{attribute 'strict'}
TYPE E_VisuCtrlPageState :
(
	SCREEN_UNINITIALIZED 		:= 0,	(*  *)
	SCREEN_INITIALIZING 		:= 1,	(*  *)
	SCREEN_READY_INITIALIZED	:= 2,	(*  *)
	SCREEN_AUTO					:= 3,	(*  *)
	SCREEN_MODE_CHANGE			:= 4,	(*  *)
	SCREEN_MANUAL_CYLINDERS		:= 5,	(*  *)
	SCREEN_MANUAL_MOTORS		:= 6,	(*  *)
	//SCREEN_MANUAL_SAFETY		:= 7,	(*  *)
	SCREEN_MANUAL_INPUTS		:= 7,	(*  *)
	SCREEN_MANUAL_OUTPUTS		:= 8,	(*  *)
	SCREEN_MANUAL_ROBOTS		:= 9,	(*  *)
	SCREEN_MANUAL_OTHERS		:= 10,	(*  *)
	SCREEN_ALARMS				:= 11,	(*  *)
	SCREEN_RECIPES				:= 12,	(*  *)
	SCREEN_RESET				:= 13,	(*  *)
	SCREEN_ABORTING				:= 14,	(*  *)
	SCREEN_EMERGENCY			:= 15	(*  *)
);
END_TYPE

(* stored: Version 1.1.0.1, ProductVersion 3.1.4024.9
   DUT E_VisuCtrlPageState: Id {1916e219-27ad-4dbd-8a52-5e082a94e0e4} *)
